// TwinCAT 3 PLC project Runtime01
// ProgramVersion: 3.1.4022.0
// libraries:
//   Tc2_Standard, * (Beckhoff Automation GmbH)
//   Tc2_System, * (Beckhoff Automation GmbH)
//   Tc3_Module, * (Beckhoff Automation GmbH)
// project tree:
//   / PlcTask.TcTTO
//   POUs/ MAIN.TcPOU

CONFIGURATION Runtime01
    RESOURCE PLC ON TwinCAT3
        TASK PlcTask(INTERVAL := T#10ms, PRIORITY := 20);
        PROGRAM MAIN WITH PlcTask : MAIN;
    END_RESOURCE
END_CONFIGURATION

// ---- POUs/MAIN.TcPOU
PROGRAM MAIN
VAR
	Temp		: LREAL;
	TempSpeed	: LREAL := 0.1;

	HeatActual	: LREAL;
	HeatSetpoint: LREAL;
	CoolActual	: LREAL;
	CoolSetpoint: LREAL;
	
	Counter	: WORD;	
	incr 	: LREAL;
	Reset		: BOOL;
END_VAR
VAR CONSTANT
	HEAT_INCR_PERSEC	: LREAL := 10;
	COOL_INCR_PERSEC	: LREAL := 3;
END_VAR

Counter := Counter + 7;

incr := HEAT_INCR_PERSEC * 1000.0 / UDINT_TO_LREAL(_TaskInfo[1].CycleTime);
HeatActual := HeatActual + SEL( HeatActual > HeatSetpoint,  incr, -incr);

incr := COOL_INCR_PERSEC * 1000.0 / UDINT_TO_LREAL(_TaskInfo[1].CycleTime);
CoolActual := CoolActual + SEL( CoolActual > CoolSetpoint,  incr, -incr);

TempSpeed := TempSpeed + 0.000007 * HeatActual - 0.000003 * CoolActual; 
Temp := Temp + TempSpeed;

IF Temp < 10 THEN
	Temp := 10;
	TempSpeed := TempSpeed / 2.0;
END_IF


IF Reset THEN
	Counter := 0;
	TempSpeed := 0;
	Temp := 0;
END_IF

END_PROGRAM
